PROGRAM POU_GatewaySignals
VAR
END_VAR

// NETWORK 1

END_PROGRAM

(* stored: Version 1.1.0.1, ProductVersion 3.1.4024.0
   POU POU_GatewaySignals: Id {bc48d4c2-b908-421e-aea4-4ea2852695f7}, SpecialFunc None *)
